TYPE U_Payload :
UNION
	sPayload : STRING(3999);
	aPayload : ARRAY[0..3999] OF BYTE;
END_UNION
END_TYPE

(* stored: Version 1.1.0.1, ProductVersion 3.1.4020.12
   DUT U_Payload: Id {d3656ed9-3c43-4b50-97c7-612023cb97c4} *)
